RESOURCE_TYPE top
  (* Standard: 61499-2 *)
  (* Version 0.1, 2017-00-25, hpea485, UOA *)
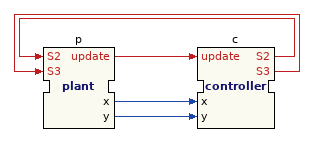
  FBS
    p : plant;
    c : controller;
  END_FBS
  EVENT_CONNECTIONS
    p.update TO c.update;
    c.S2 TO p.S2;
    c.S3 TO p.S3;
  END_CONNECTIONS
  DATA_CONNECTIONS
    p.x TO c.x;
    p.y TO c.y;
  END_CONNECTIONS
END_RESOURCE_TYPE
